INTERFACE I_PersistentEventStorage

METHOD StoreEvent
VAR_INPUT
	stEvent : ST_Event;
END_VAR
END_METHOD

END_INTERFACE

(* stored: Version 1.1.0.1, ProductVersion 3.1.4024.12
   Itf I_PersistentEventStorage: Id {6a7c310f-6b2e-4b18-9621-5a462b180780}
   Method StoreEvent: Id {d071ed3f-4cbe-42d9-908d-aaa66b46b5b2} *)
